PROGRAM PRG_ReadTime
VAR 
	//Delta time in ms from Digital sensor to camera TCP
	aDeltaTimeMS			: ARRAY[0..GVL_Constant.ITEM_ARRAY_SIZE] OF UDINT;

	//Digital input sensor
	aDigitalSensorTime		: ARRAY[0..ITEM_ARRAY_SIZE] OF STRING;
	
	//Camera TCP port
	aTCPPortCameraTime	:ARRAY[0..ITEM_ARRAY_SIZE] OF STRING;
	
END_VAR


SaveSensorTime();
SaveCameraTCPTime();
CalculateDeltaTime();

METHOD PUBLIC CalculateDeltaTime
VAR
	iDeltaTime			:INT;
	iNDeltaTime			:INT;
	rDeltaTrig			:R_TRIG;
	SavedCameraTime		:T_FILETIME;
	SavedSensorTime		:T_FILETIME;
	
END_VAR
//Get saved time from camera and sensor method
SavedCameraTime:=SaveCameraTCPTime();
SavedSensorTime:=SaveSensorTime();

//Trigger of camera tcp read complete. Uses same as camera as this is the last one to receive
rDeltaTrig(CLK:=PRG_TCPIP.fbReadFromCameraTCP.bReadComplete);

IF rDeltaTrig.Q THEN
	
	//Calculate delta time
	aDeltaTimeMS[iDeltaTime] :=  (F_CXSubTimeStamp(nTimeStampHiDW_A:=SavedCameraTime.dwHighDateTime,
													   nTimeStampHiDW_B:=SavedSensorTime.dwHighDateTime,
													   nTimeStampLoDW_A:=SavedCameraTime.dwLowDateTime,
													   nTimeStampLoDW_B:=SavedSensorTime.dwLowDateTime)/1000);
	iDeltaTime := iDeltaTime +1;
END_IF

//Reset registry
IF GVL_Timestamp.bResetRegistry THEN
	FOR iNDeltaTime := 0 TO GVL_Constant.ITEM_ARRAY_SIZE DO 
		aDeltaTimeMS[iNDeltaTime] := 0;
	END_FOR
	iDeltaTime := 0;
END_IF
END_METHOD

METHOD PUBLIC SaveCameraTCPTime : T_FILETIME
VAR
	rTCPPortCamera		:R_TRIG;
	iTCPPortCamera		:INT;
	iNTCPCamera			:INT;
	fbGetCameraTime		:FB_SystemTime;
END_VAR
//Trigger of camera tcp read complete
rTCPPortCamera(CLK:=PRG_TCPIP.fbReadFromCameraTCP.bReadComplete);

IF rTCPPortCamera.Q THEN
	aTCPPortCameraTime[iTCPPortCamera] := fbGetCameraTime.M_SystemTimeToString();
	
	fbGetCameraTime.fbSystemTime(timeLoDW=>SaveCameraTCPTime.dwLowDateTime,
    							 timeHiDW=>SaveCameraTCPTime.dwHighDateTime);
	
	iTCPPortCamera := iTCPPortCamera +1;
END_IF

//Reset registry
IF GVL_Timestamp.bResetRegistry THEN
	FOR iNTCPCamera := 0 TO GVL_Constant.ITEM_ARRAY_SIZE DO 
		aTCPPortCameraTime[iNTCPCamera] := '';
	END_FOR
	iTCPPortCamera := 0;
END_IF
END_METHOD

METHOD PUBLIC SaveSensorTime : T_FILETIME
VAR
	rDigitalSensorIn		:R_TRIG;
	iDigitalSensor			:INT;
	iNDigitalSensor			:INT;
	fbGetSensorTime			:FB_SystemTime;
END_VAR
//Trigger of sensor input
rDigitalSensorIn(CLK:=GVL_ItemSimulator.bSignalIn);

IF rDigitalSensorIn.Q THEN
	aDigitalSensorTime[iDigitalSensor] := fbGetSensorTime.M_SystemTimeToString();
	
	fbGetSensorTime.fbSystemTime(timeLoDW=>SaveSensorTime.dwLowDateTime,
    							 timeHiDW=>SaveSensorTime.dwHighDateTime);
								 
	iDigitalSensor := iDigitalSensor +1;
END_IF

//Reset registry
IF GVL_Timestamp.bResetRegistry THEN
	FOR iNDigitalSensor := 0 TO GVL_Constant.ITEM_ARRAY_SIZE DO 
		aDigitalSensorTime[iNDigitalSensor] := '';
	END_FOR
	iDigitalSensor := 0;
END_IF
END_METHOD

END_PROGRAM

(* stored: Version 1.1.0.1, ProductVersion 3.1.4024.12
   POU PRG_ReadTime: Id {41809a93-5b53-47f0-b8b5-05c700b2cea3}, SpecialFunc None
   Method CalculateDeltaTime: Id {a5129a3c-0d36-4a82-bf14-e117a70e330a}
   Method SaveCameraTCPTime: Id {9f3cdf40-e788-4c90-aed5-163aedc53860}
   Method SaveSensorTime: Id {cd1a26d1-d744-4b0d-8d44-8a38ddfb04e9} *)
